FUNCTION_BLOCK TcoDesignerTrigger_v_2_x_x EXTENDS TcoCore.TcoTask
VAR_INPUT
	inTriggerType:eTcoDesignerTriggerType;
	refClearResultsTask: REFERENCE TO TcoDesignerClearInspectionResults_v_2_x_x;
END_VAR 

VAR
	_clearResultsTask: REFERENCE TO TcoDesignerClearInspectionResults_v_2_x_x;
END_VAR
VAR_IN_OUT
	inoIoData	: TcoDesignerData_2_x_x;
    inoConfig	: TcoDesignerConfig_v_2_x_x;
	inoStatus	: TcoDesignerStatus_v_2_x_x;	
	//inoResults	: TcoInsightResults_v_5_x_x;
END_VAR
VAR
   
	_progress : INT := 0;
    {attribute 'hide'} 
	_infoTimer :  TON;
    {attribute 'hide'} 
	_errorTimer :  TON;
    {attribute 'hide'} 
	_varInfo : __SYSTEM.VAR_INFO;
    {attribute 'hide'} 
	_sb : TcoCore.StringBuilder;
  
END_VAR

IF NOT __ISVALIDREF(refClearResultsTask)  THEN
    Messenger.Post('<#Invalid reference ClearResultsTask>', TcoCore.eMessageCategory.ProgrammingError);
    RETURN;
END_IF
_clearResultsTask REF= refClearResultsTask;

IF Execute() THEN
	IF _progress = 0 THEN
		IF NOT __ISVALIDREF(inoIoData) THEN
			_varInfo :=__VARINFO(inoIoData);
			Messenger.Programming(_sb.Clear().Append('<#Invalid reference: #>').Append(_varInfo.Symbol).ToString()).Pin();
		ELSIF NOT __ISVALIDREF(inoConfig) THEN                                                  
			_varInfo :=__VARINFO(inoConfig);                                                    
			Messenger.Programming(_sb.Clear().Append('<#Invalid reference: #>').Append(_varInfo.Symbol).ToString()).Pin();
		ELSIF NOT __ISVALIDREF(inoStatus) THEN                                                  
			_varInfo :=__VARINFO(inoStatus);                                                    
			Messenger.Programming(_sb.Clear().Append('<#Invalid reference: #>').Append(_varInfo.Symbol).ToString()).Pin();

		ELSIF inTriggerType = eTcoDesignerTriggerType.TriggerWithTimeout 
			AND inoConfig.ErrorTime < inoConfig.TriggerTimemout  AND inoConfig.ErrorTime <>T#0S THEN
				Messenger.Error(_sb.Clear().Append('<#Error time is lower than timeout. Please check config!#>').ToString()).Pin();

		ELSE
			_progress := _progress + 1;
			CallTimers(FALSE);

		END_IF
	END_IF
	
		
	IF _progress = 1 THEN
		IF inTriggerType = eTcoDesignerTriggerType.TriggerFast THEN
			_progress := _progress + 1;
		ELSIF inTriggerType = eTcoDesignerTriggerType.TriggerWithTimeout THEN
			inoIoData.PlcToPc.Timeout:=TIME_TO_UINT( inoConfig.TriggerTimemout);
			IF _clearResultsTask.Invoke().Done THEN
				_progress := _progress + 1;
			END_IF;
		ELSIF _clearResultsTask.Invoke().Done THEN
			_progress := _progress + 1;
		END_IF

	END_IF;
	
	IF _progress = 2 THEN
		THIS^.Messenger.OnCondition(_infoTimer.Q).Warning('<#Waiting for the Online signal!#>'); 
		IF THIS^.inoIoData.PcToPlc.SystemOnline THEN
			CallTimers(FALSE);
			_progress := _progress + 1;
		END_IF
	END_IF
	

	IF _progress = 3 THEN
		THIS^.Messenger.OnCondition(_infoTimer.Q).Info('<#Trigger!#>'); 
		THIS^.inoIoData.PlcToPc.Trigger:=TRUE;
	
		IF NOT THIS^.inoIoData.PcToPlc.InspectionReady  THEN
			THIS^.inoIoData.PlcToPc.Trigger:=FALSE;
			CallTimers(FALSE);
			_progress := _progress + 1;
		END_IF
	END_IF
	
	
	IF _progress=4 THEN	
		Messenger.Info('Waiting for results available');
		IF THIS^.inoIoData.PcToPlc.ResultsAvailable  THEN		
			CallTimers(FALSE);
			_progress := _progress + 1;
		END_IF
	END_IF
	
	IF _progress=5 THEN	
		Messenger.Info('Acknovledge results');
		THIS^.inoIoData.PlcToPc.ResultsAck:=TRUE;
		IF NOT THIS^.inoIoData.PcToPlc.ResultsAvailable  THEN
			THIS^.inoIoData.PlcToPc.ResultsAck:=FALSE;
			THIS^.DoneWhen(TRUE);
			
		END_IF
	END_IF
	

	

	CallTimers(TRUE);
	
	THIS^.ThrowWhen(_errorTimer.Q  OR THIS^.inoIoData.PcToPlc.Error 
		OR (inTriggerType = eTcoDesignerTriggerType.TriggerWithTimeout AND THIS^.inoIoData.PcToPlc.TriggerTimeout) );	

END_IF

METHOD CallTimers
VAR_INPUT
	inValue : BOOL;
END_VAR
IF  __ISVALIDREF(inoConfig) AND THIS^.inoConfig.ErrorTime <> T#0S OR NOT inValue THEN  
_errorTimer(IN := inValue, PT := THIS^.inoConfig.ErrorTime);
END_IF;
IF  __ISVALIDREF(inoConfig) AND THIS^.inoConfig.InfoTime <>T#0S OR NOT inValue THEN  
_infoTimer(IN := inValue, PT := THIS^.inoConfig.InfoTime);
END_IF;
END_METHOD

(*~
	<docu>
		<summary>
			Executes when task is aborted.
		</summary>			
	</docu>	
~*)
METHOD PROTECTED OnAbort
THIS^.inoStatus.ActionDescription := '<#Trigger was aborted, while not yet completed!#>';
END_METHOD

(*~
	<docu>
		<summary>
			Executes when task reaches the ```Done``` state .
		</summary>			
	</docu>	
~*)
METHOD PROTECTED OnDone
THIS^.inoStatus.ActionDescription := '<#Trigger was completed successfully.#>'; 
_progress:=0;
END_METHOD

(*~
	<docu>
		<summary>
			Executes when task reaches the ```Error``` state.
			<para>
				Do not confuse with <see cref="PlcDocu.TcoCore.TcoTask.WhileError()"/>, that is called cyclically until '''Error''' state is left.
			</para>
		</summary>			
	</docu>	
~*)
METHOD PROTECTED OnError
THIS^.inoStatus.ActionDescription := '<#Trigger finished with error.#>';
END_METHOD

METHOD PROTECTED OnStart
THIS^.inoStatus.ActionDescription := '<#Trigger started.#>'; 
inoIoData.PlcToPc.Timeout:=0;
END_METHOD

(*~
	<docu>
		<summary>
			Restores this instance to the Ready state. Can be called explicitly or from within one of the restore mechanisms.
			<para>
				See also <see cref="PlcDocu.TcoCore.TcoTask.AutoRestorable()"/>
			</para>
		</summary>			
	</docu>	
~*)
METHOD Restore : ITcoRestorable
SUPER^.Restore();
_progress := 0;
CallTimers(FALSE);
Messenger.UnPin();
END_METHOD

END_FUNCTION_BLOCK

(* stored: Version 1.1.0.1, ProductVersion 3.1.4024.12
   POU TcoDesignerTrigger_v_2_x_x: Id {34c24828-75cb-0fee-06b4-7614eae7d9e2}, SpecialFunc None
   Method CallTimers: Id {b7ec5859-98ed-009d-331f-b2e23cb1dcfd}
   Method OnAbort: Id {fee7fe37-7d09-0a35-3b6e-db34c6b40ed8}
   Method OnDone: Id {27498230-0e21-074c-3591-33b08904246e}
   Method OnError: Id {409e6e93-f502-0b75-318d-4b1126b27ae7}
   Method OnStart: Id {1b979094-8bfb-0136-3823-7af7f9cc07cb}
   Method Restore: Id {05ef5298-f98e-091a-21f3-c18438677618} *)
